FUNCTION_BLOCK Basic (* Basic Function Block Type *)
  (* Standard: 61499-2 *)
  (* Version 0.2, 2003-12-04, JHC, Rockwell Automation, Renamed for better indexing. *)
  (* Version 0.1, 2002-11-05, JHC, Rockwell Automation, Corrected missing ST element in Algorithm REQ. *)
  (* Version 0.0, 2000-05-30, JHC, Rockwell Automation *)
  (* Compiler header: package fb.rt.template; *)
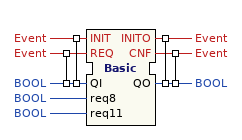
  EVENT_INPUT
    INIT WITH QI, NOTQI; (* Initialization Request *)
    REQ WITH QI, NOTQI; (* Normal Execution Request *)
  END_EVENT
  EVENT_OUTPUT
    INITO WITH QO; (* Initialization Confirm *)
    CNF WITH QO; (* Execution Confirmation *)
  END_EVENT
  VAR_INPUT
    QI : BOOL; (* Input event qualifier *)
    req8 : BOOL;
    req11 : BOOL;
  END_VAR
  VAR_OUTPUT
    QO : BOOL;
  END_VAR
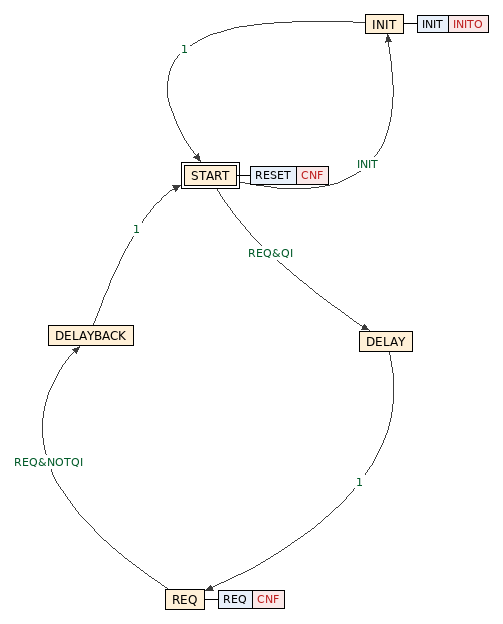
  EC_STATES
    START : RESET -> CNF; (* Initial State *)
    INIT : INIT -> INITO; (* Initialization *)
    REQ : REQ -> CNF; (* Normal execution *)
    DELAY;
    DELAYBACK;
  END_STATES
  EC_TRANSITIONS
    START TO INIT := INIT;
    INIT TO START := 1;
    DELAY TO REQ := 1;
    START TO DELAY := REQ&QI;
    DELAYBACK TO START := 1;
    REQ TO DELAYBACK := REQ&NOTQI;
  END_TRANSITIONS
  ALGORITHM INIT IN ST: (* Initialization algorithm *)

  END_ALGORITHM
  ALGORITHM REQ IN Java: (* Normally executed algorithm *)
QO.value = true;
  END_ALGORITHM
  ALGORITHM RESET IN Java:
QO.value = false;
  END_ALGORITHM
END_FUNCTION_BLOCK
